FUNCTION_BLOCK FB_CNC_MILL
VAR_INPUT
	IN : BOOL;
	Opened	: BOOL;
	Busy	: BOOL;
	Error	: BOOL;
	mProgress : WORD;
END_VAR
VAR_OUTPUT
	Q		: BOOL;
	Start	: BOOL;
	Stop	: BOOL;
	Reset	: BOOL;
	Produce_Lids_Or_Dont	: BOOL;
END_VAR
VAR
	iState: INT;
END_VAR

IF NOT IN THEN
	Q := 		FALSE;
	Start := 	FALSE;
	ELSE
		Q := 		TRUE;
		Start := 	TRUE;
END_IF

END_FUNCTION_BLOCK

(* stored: Version 1.1.0.1, ProductVersion 3.1.4024.6
   POU FB_CNC_MILL: Id {0619a382-ef17-4bd0-9cc7-f203258ebcd1}, SpecialFunc None *)
